Staubli VAL3: OnF7.pgx

program OnF7()
begin
  //
  PublicData:bSimulaiton=false
  call Motion:AllMotion(PublicData:sStartPrd)
  PublicData:libSave()
  bUserRefresh=true
end
